// TIA Portal V19 export
DATA_BLOCK "PPrgArchive10"   // DB503
// stored: IsOnlyStoredInLoadMemory true, MemoryReserve 0, Namespace G
   VAR RETAIN
      PRG : Array[901..1000] of "PPrg_Data";
   END_VAR
BEGIN
END_DATA_BLOCK
